// TIA Portal V18 export
DATA_BLOCK "Function Dearing with valve"   // DB46
{ S7_Optimized_Access := 'TRUE' }
VERSION : 0.1
// stored: AutoNumber true, DBAccessibleFromOPCUA true, IsOnlyStoredInLoadMemory false, IsRetainMemResEnabled false, IsWriteProtectedInAS false, MemoryReserve 100
   VAR RETAIN
      "Input A" : Struct
         "set time" : Int;
         "set flowrate" : Real;
      END_STRUCT;
      "Input B" : Struct
         "set time" : Int;
         "set flowrate" : Real;
      END_STRUCT;
   END_VAR
   VAR
      "Control A" : Struct
         "start deaaring" : Bool;
         "dearing running" : Bool;
         "stop dearing" : Bool;
         "dearing Completed" : Bool;
      END_STRUCT;
      "Control B" : Struct
         "start deaaring" : Bool;
         "dearing running" : Bool;
         "stop dearing" : Bool;
         "dearing Completed" : Bool;
      END_STRUCT;
      "Output A" : Struct
         "ON pump" : Bool;
         "On outlet valve" : Bool;
         "running time" : Int;
         "ON_inlet A" : Bool;
      END_STRUCT;
      "Output B" : Struct
         "ON pump" : Bool;
         "running time" : Int;
         "On outlet valve" : Bool;
         "ON_inlet B" : Bool;
      END_STRUCT;
   END_VAR
   VAR RETAIN
      "start signal Type" : Int;
   END_VAR
BEGIN
END_DATA_BLOCK
